FUNCTION_BLOCK FB_InfoGroup
VAR_INPUT
	stInfoData	:ST_InfoDataGroup;
END_VAR
VAR_OUTPUT
	sState		:STRING;
END_VAR
VAR
END_VAR

IF stInfoData.usiMapState= 1 THEN
	sState:='RUN';
ELSIF stInfoData.usiMapState= 2 THEN
	sState:='STOP';
ELSIF stInfoData.usiMapState= 3 THEN
	sState:='SAFE';
ELSIF stInfoData.usiMapState= 4 THEN
	sState:='ERROR';
ELSIF stInfoData.usiMapState= 5 THEN
	sState:='RESET';
ELSE
	sState:='Unknown';
END_IF

END_FUNCTION_BLOCK

(* stored: Version 1.1.0.1, ProductVersion 3.1.4024.12
   POU FB_InfoGroup: Id {47978db8-33aa-4916-84ea-dd7136349c3d}, SpecialFunc None *)
